TYPE ST_ControlElement_HMI EXTENDS ST_BaseControlElement_HMI :
STRUCT
	
END_STRUCT
END_TYPE

(* stored: Version 1.1.0.1, ProductVersion 3.1.4024.15
   DUT ST_ControlElement_HMI: Id {2058c532-d1b3-450f-a008-e980fa54748a} *)
